{attribute 'qualified_only'}
VAR_GLOBAL
END_VAR

(* stored: Version 1.1.0.1, ProductVersion 3.1.4022.7
   GVL GVL_05_Manual_Step_Motor_BOX_Y: Id {746c4302-0407-426a-a496-81551dbbf0eb} *)
